TEXTLIST WorkAreaTypology
  0 = '-'
  1 = 'Pallet (Magazine)'
  2 = 'Pallet (Work)'
  3 = 'Layer (Magazine)'
   = ''
END_TEXTLIST

(* stored: Version 1.1.0.1, ProductVersion 3.1.4024.11
   TextList WorkAreaTypology: Id {47745bb4-69f0-4a35-aff8-eae24eaf7814} *)
